TYPE ST_BufferControl :
STRUCT
	stData			: ST_MMBuffer;		// Data for vehicle
	iMoveCmdID		: UINT;				// Command ID for movement (to check status for movement)
END_STRUCT
END_TYPE

(* stored: Version 1.1.0.1, ProductVersion 3.1.4024.5
   DUT ST_BufferControl: Id {4cb5bb87-0c0d-4ad6-b44e-91f223606e94} *)
